FUNCTION_BLOCK Module_call
VAR_INPUT
END_VAR
VAR_OUTPUT
END_VAR
VAR
	CC1_UNIT1_3_Cyl: FB_CylinderModule;	
	CC2_UNIT2_3_Cyl: FB_CylinderModule;
	CC3_UNIT3_3_Cyl: FB_CylinderModule;
	CC4_UNIT4_3_Cyl: FB_CylinderModule;
	CC5_UNIT5_1_Cyl: FB_CylinderModule;
	CC6_UNIT6_1_Cyl: FB_CylinderModule;
	CC1_Feedback_FB: Feedback_FB;
	CC2_Feedback_FB: Feedback_FB;
	CC3_Feedback_FB: Feedback_FB;
	CC4_Feedback_FB: Feedback_FB;
	CC5_Feedback_FB: Feedback_FB;
	CC6_Feedback_FB: Feedback_FB;
	CC1_Feedback_1: BOOL;
	CC1_Feedback_2: BOOL;
	CC2_Feedback_1: BOOL;
	CC2_Feedback_2: BOOL;
	CC3_Feedback_1: BOOL;
	CC3_Feedback_2: BOOL;
	CC4_Feedback_1: BOOL;
	CC4_Feedback_2: BOOL;
	PowerOn: PowerOn;
	TurnTable_0: TurnTable;
	TT_Feedback_FB: Feedback_FB;
	Trunion_0: Trunion;
	Tr_Feedback_FB: Feedback_FB;
	RollerDoor_0: RollerDoor;
	Door_Feedback_FB: Feedback_FB;
	MH_Robot: Robot;
	Weld_Robot: Robot;
	Auto_Sequence_0: Auto_Sequence;
	TR_Feedback_FB1: Feedback_FB;
	HomeSequence_0: HomeSequence;
	Alarms_0: Alarms;
END_VAR
VAR // added by the converter: edge detectors and wires of the graphical bodies
    _w1, _w2, _w3, _w4, _w5, _w6, _w7, _w8 : BOOL;
END_VAR

// note: this text did not pass the execution check against the stored diagram
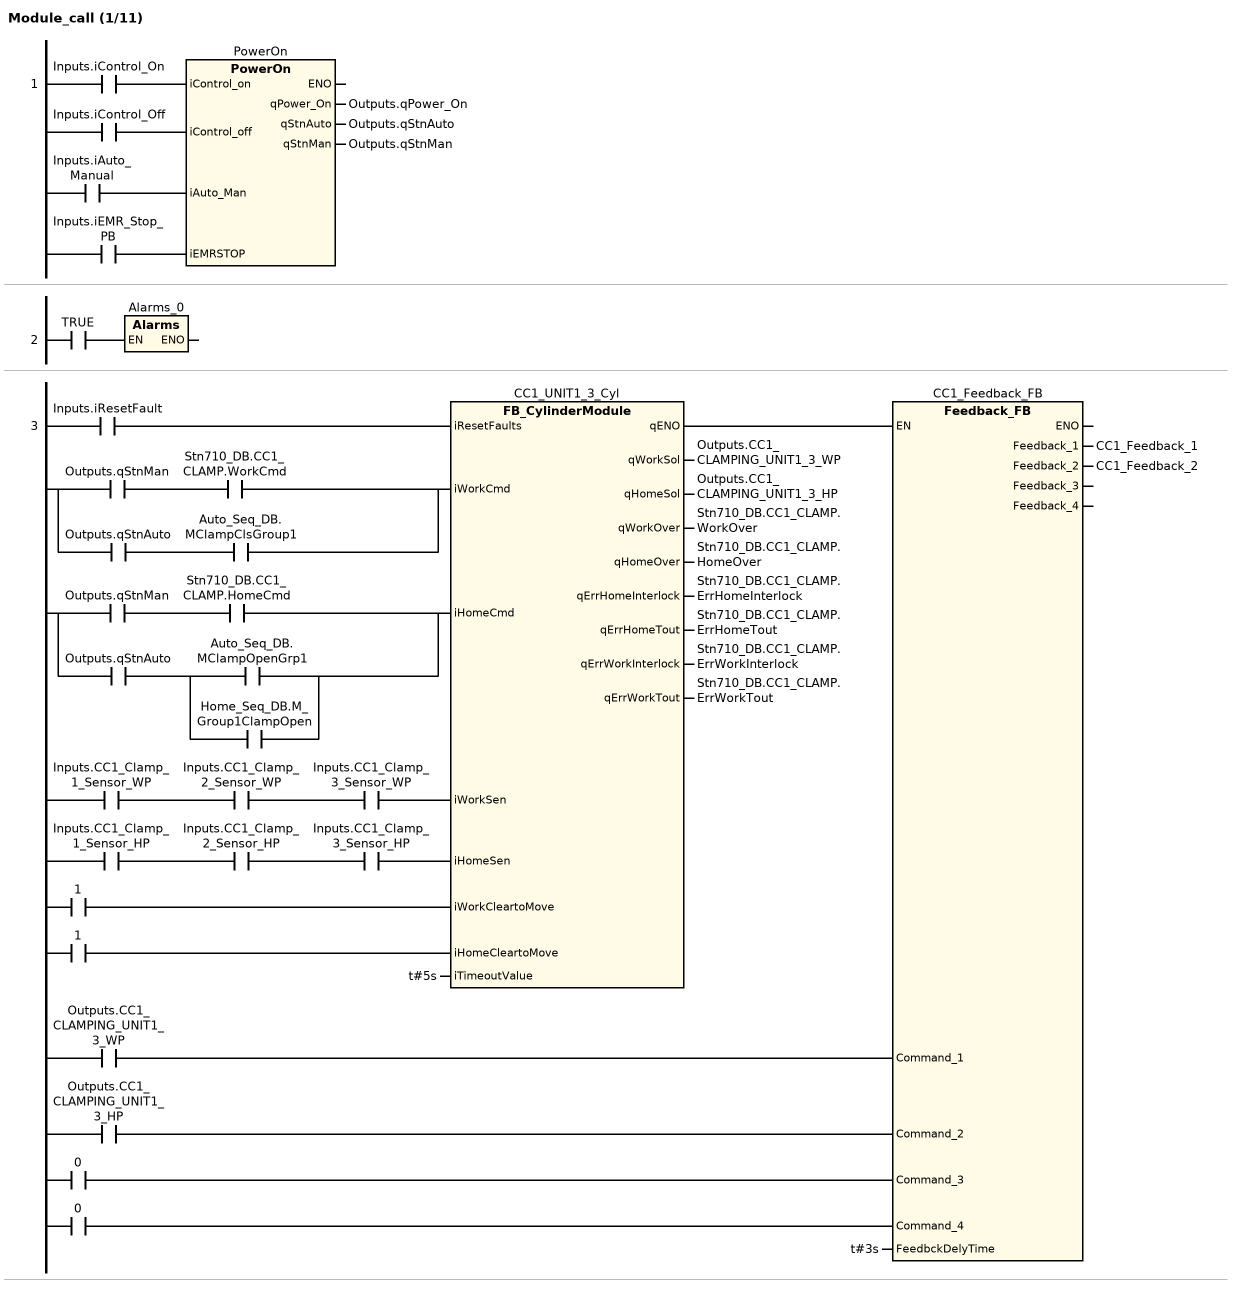
// NETWORK 1
PowerOn(
    iControl_on := Inputs.iControl_On,
    iControl_off := Inputs.iControl_Off,
    iAuto_Man := Inputs.iAuto_Manual,
    iEMRSTOP := Inputs.iEMR_Stop_PB,
    qPower_On => Outputs.qPower_On,
    qStnAuto => Outputs.qStnAuto,
    qStnMan => Outputs.qStnMan);

// NETWORK 2
Alarms_0(EN := TRUE); // Alarms

// NETWORK 3
CC1_UNIT1_3_Cyl(
    iResetFaults := Inputs.iResetFault,
    iWorkCmd := Outputs.qStnMan AND Stn710_DB.CC1_CLAMP.WorkCmd OR Outputs.qStnAuto AND Auto_Seq_DB.MClampClsGroup1,
    iHomeCmd := Outputs.qStnMan AND Stn710_DB.CC1_CLAMP.HomeCmd OR Outputs.qStnAuto AND (Auto_Seq_DB.MClampOpenGrp1 OR Home_Seq_DB.M_Group1ClampOpen),
    iWorkSen := Inputs.CC1_Clamp_1_Sensor_WP AND Inputs.CC1_Clamp_2_Sensor_WP AND Inputs.CC1_Clamp_3_Sensor_WP,
    iHomeSen := Inputs.CC1_Clamp_1_Sensor_HP AND Inputs.CC1_Clamp_2_Sensor_HP AND Inputs.CC1_Clamp_3_Sensor_HP,
    iWorkCleartoMove := 1,
    iHomeCleartoMove := 1,
    iTimeoutValue := t#5s,
    qWorkSol => Outputs.CC1_CLAMPING_UNIT1_3_WP,
    qHomeSol => Outputs.CC1_CLAMPING_UNIT1_3_HP,
    qWorkOver => Stn710_DB.CC1_CLAMP.WorkOver,
    qHomeOver => Stn710_DB.CC1_CLAMP.HomeOver,
    qErrHomeInterlock => Stn710_DB.CC1_CLAMP.ErrHomeInterlock,
    qErrHomeTout => Stn710_DB.CC1_CLAMP.ErrHomeTout,
    qErrWorkInterlock => Stn710_DB.CC1_CLAMP.ErrWorkInterlock,
    qErrWorkTout => Stn710_DB.CC1_CLAMP.ErrWorkTout); // FB_CylinderModule
CC1_Feedback_FB(
    EN := CC1_UNIT1_3_Cyl.qENO,
    Command_1 := Outputs.CC1_CLAMPING_UNIT1_3_WP,
    Command_2 := Outputs.CC1_CLAMPING_UNIT1_3_HP,
    Command_3 := 0,
    Command_4 := 0,
    FeedbckDelyTime := t#3s,
    Feedback_1 => CC1_Feedback_1,
    Feedback_2 => CC1_Feedback_2); // Feedback_FB

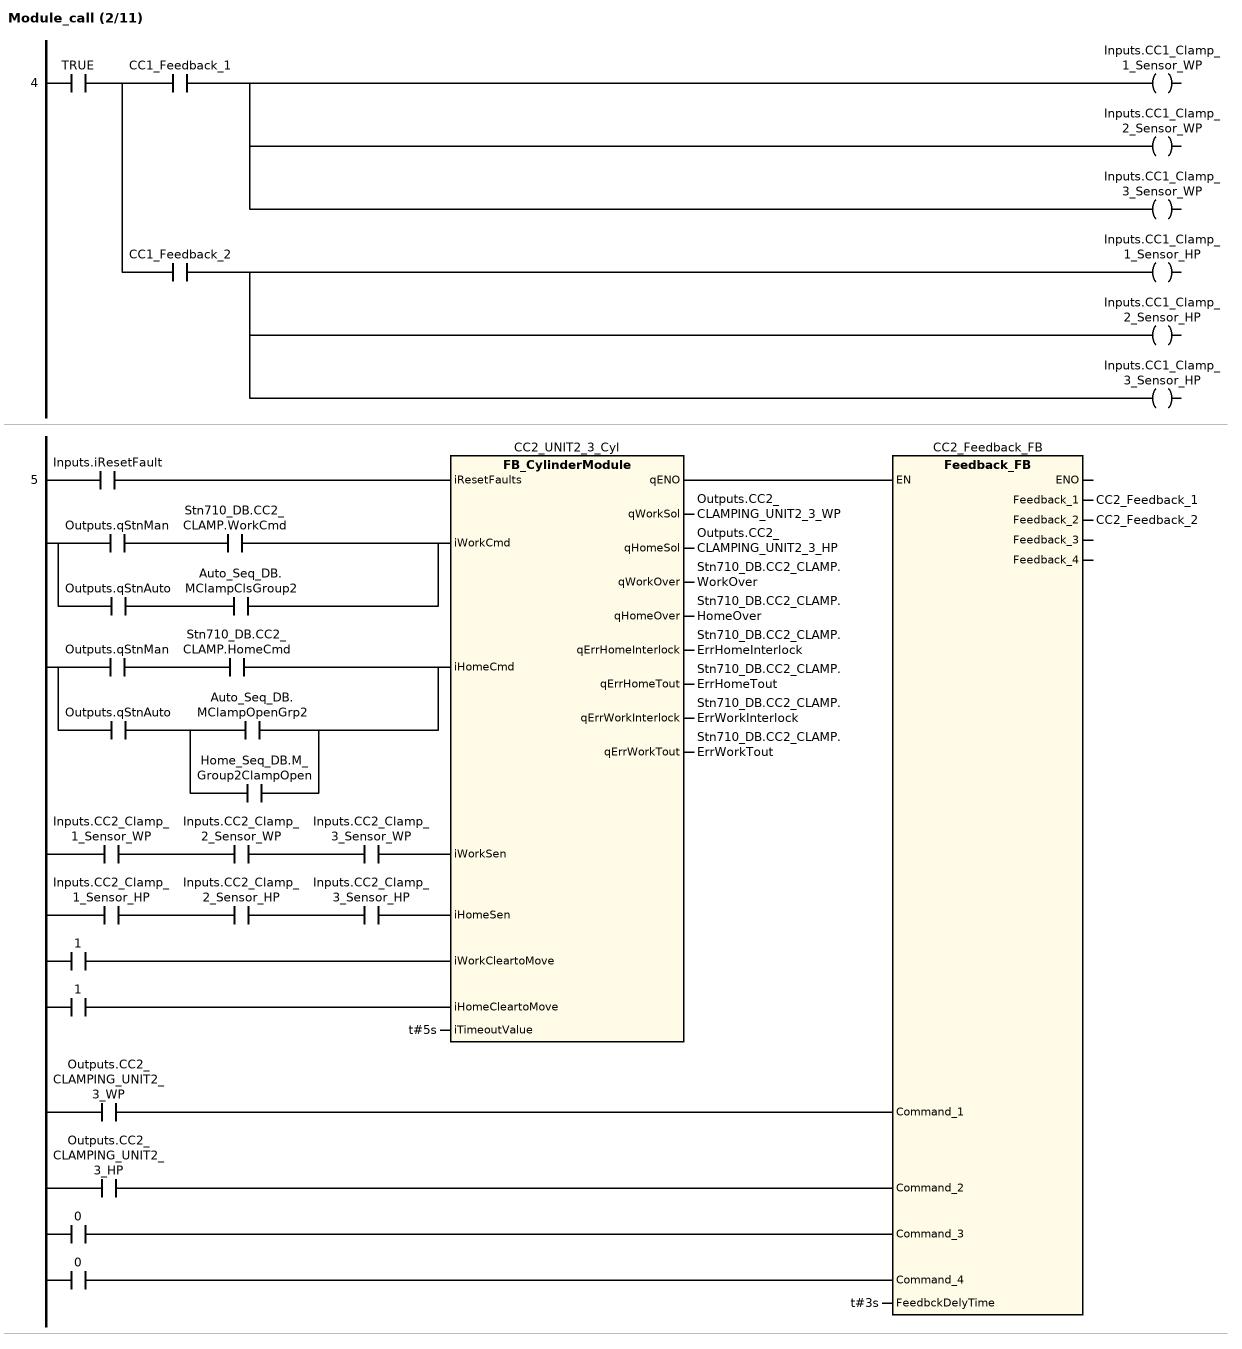
// NETWORK 4
_w1 := TRUE AND CC1_Feedback_1;
Inputs.CC1_Clamp_1_Sensor_WP := _w1;
Inputs.CC1_Clamp_2_Sensor_WP := _w1;
Inputs.CC1_Clamp_3_Sensor_WP := _w1;
_w2 := TRUE AND CC1_Feedback_2;
Inputs.CC1_Clamp_1_Sensor_HP := _w2;
Inputs.CC1_Clamp_2_Sensor_HP := _w2;
Inputs.CC1_Clamp_3_Sensor_HP := _w2;

// NETWORK 5
CC2_UNIT2_3_Cyl(
    iResetFaults := Inputs.iResetFault,
    iWorkCmd := Outputs.qStnMan AND Stn710_DB.CC2_CLAMP.WorkCmd OR Outputs.qStnAuto AND Auto_Seq_DB.MClampClsGroup2,
    iHomeCmd := Outputs.qStnMan AND Stn710_DB.CC2_CLAMP.HomeCmd OR Outputs.qStnAuto AND (Auto_Seq_DB.MClampOpenGrp2 OR Home_Seq_DB.M_Group2ClampOpen),
    iWorkSen := Inputs.CC2_Clamp_1_Sensor_WP AND Inputs.CC2_Clamp_2_Sensor_WP AND Inputs.CC2_Clamp_3_Sensor_WP,
    iHomeSen := Inputs.CC2_Clamp_1_Sensor_HP AND Inputs.CC2_Clamp_2_Sensor_HP AND Inputs.CC2_Clamp_3_Sensor_HP,
    iWorkCleartoMove := 1,
    iHomeCleartoMove := 1,
    iTimeoutValue := t#5s,
    qWorkSol => Outputs.CC2_CLAMPING_UNIT2_3_WP,
    qHomeSol => Outputs.CC2_CLAMPING_UNIT2_3_HP,
    qWorkOver => Stn710_DB.CC2_CLAMP.WorkOver,
    qHomeOver => Stn710_DB.CC2_CLAMP.HomeOver,
    qErrHomeInterlock => Stn710_DB.CC2_CLAMP.ErrHomeInterlock,
    qErrHomeTout => Stn710_DB.CC2_CLAMP.ErrHomeTout,
    qErrWorkInterlock => Stn710_DB.CC2_CLAMP.ErrWorkInterlock,
    qErrWorkTout => Stn710_DB.CC2_CLAMP.ErrWorkTout); // FB_CylinderModule
CC2_Feedback_FB(
    EN := CC2_UNIT2_3_Cyl.qENO,
    Command_1 := Outputs.CC2_CLAMPING_UNIT2_3_WP,
    Command_2 := Outputs.CC2_CLAMPING_UNIT2_3_HP,
    Command_3 := 0,
    Command_4 := 0,
    FeedbckDelyTime := t#3s,
    Feedback_1 => CC2_Feedback_1,
    Feedback_2 => CC2_Feedback_2); // Feedback_FB

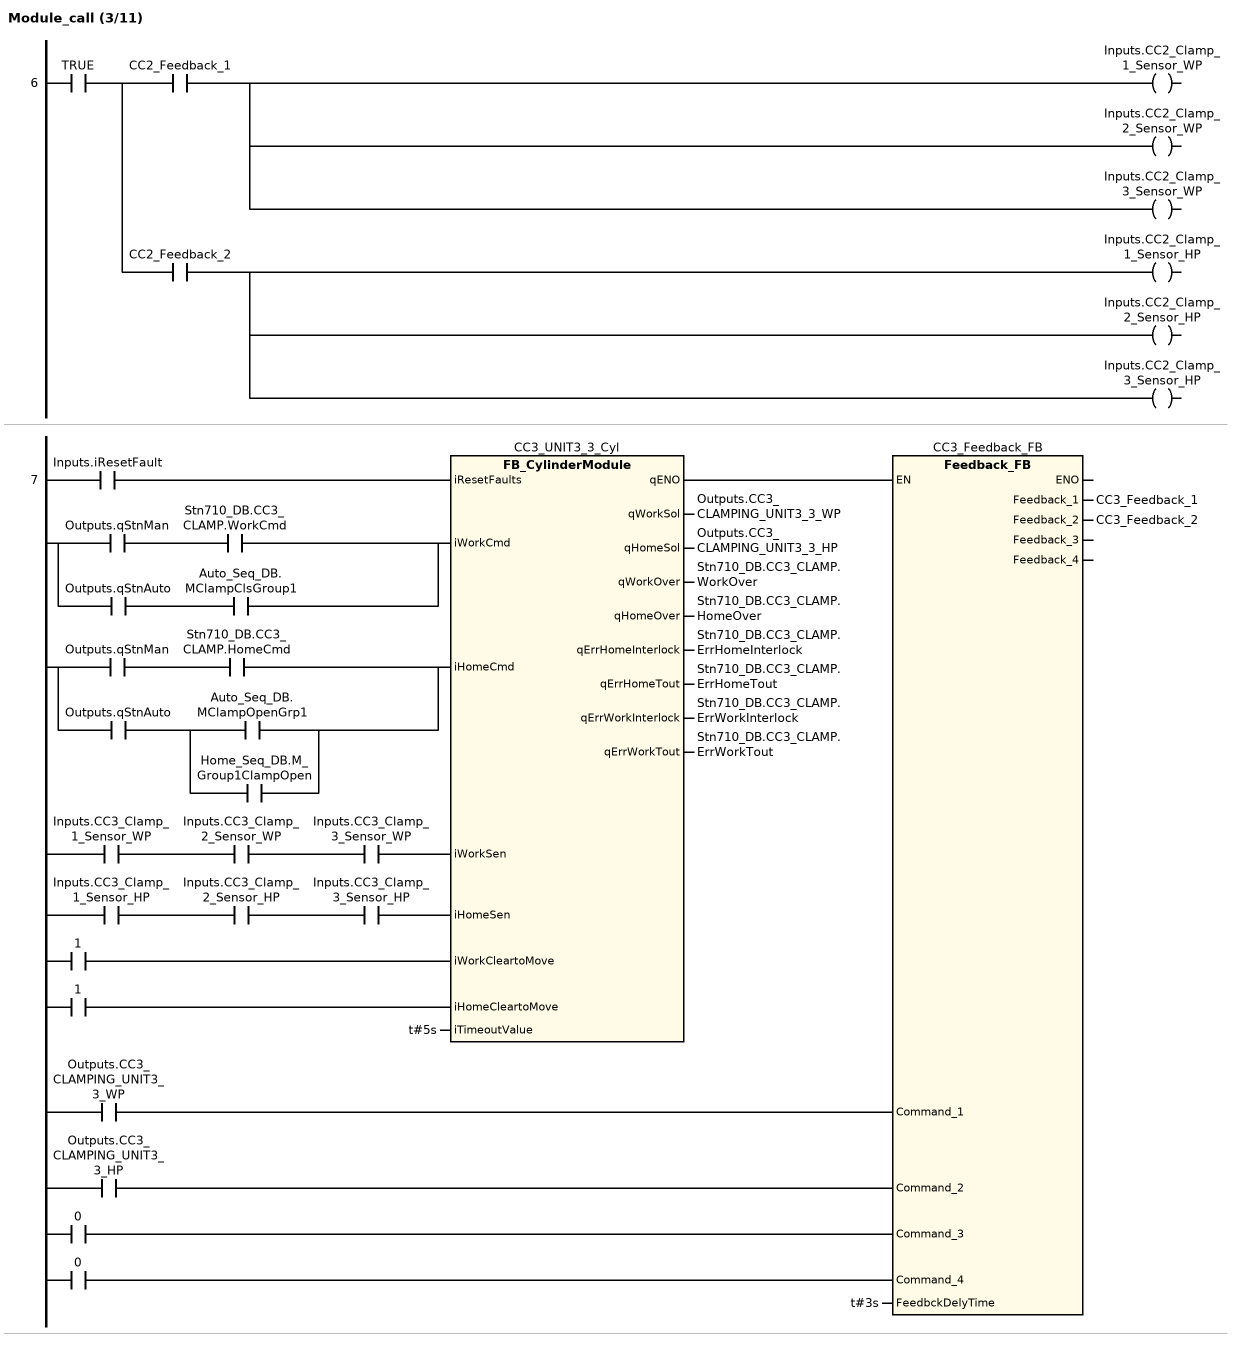
// NETWORK 6
_w3 := TRUE AND CC2_Feedback_1;
Inputs.CC2_Clamp_1_Sensor_WP := _w3;
Inputs.CC2_Clamp_2_Sensor_WP := _w3;
Inputs.CC2_Clamp_3_Sensor_WP := _w3;
_w4 := TRUE AND CC2_Feedback_2;
Inputs.CC2_Clamp_1_Sensor_HP := _w4;
Inputs.CC2_Clamp_2_Sensor_HP := _w4;
Inputs.CC2_Clamp_3_Sensor_HP := _w4;

// NETWORK 7
CC3_UNIT3_3_Cyl(
    iResetFaults := Inputs.iResetFault,
    iWorkCmd := Outputs.qStnMan AND Stn710_DB.CC3_CLAMP.WorkCmd OR Outputs.qStnAuto AND Auto_Seq_DB.MClampClsGroup1,
    iHomeCmd := Outputs.qStnMan AND Stn710_DB.CC3_CLAMP.HomeCmd OR Outputs.qStnAuto AND (Auto_Seq_DB.MClampOpenGrp1 OR Home_Seq_DB.M_Group1ClampOpen),
    iWorkSen := Inputs.CC3_Clamp_1_Sensor_WP AND Inputs.CC3_Clamp_2_Sensor_WP AND Inputs.CC3_Clamp_3_Sensor_WP,
    iHomeSen := Inputs.CC3_Clamp_1_Sensor_HP AND Inputs.CC3_Clamp_2_Sensor_HP AND Inputs.CC3_Clamp_3_Sensor_HP,
    iWorkCleartoMove := 1,
    iHomeCleartoMove := 1,
    iTimeoutValue := t#5s,
    qWorkSol => Outputs.CC3_CLAMPING_UNIT3_3_WP,
    qHomeSol => Outputs.CC3_CLAMPING_UNIT3_3_HP,
    qWorkOver => Stn710_DB.CC3_CLAMP.WorkOver,
    qHomeOver => Stn710_DB.CC3_CLAMP.HomeOver,
    qErrHomeInterlock => Stn710_DB.CC3_CLAMP.ErrHomeInterlock,
    qErrHomeTout => Stn710_DB.CC3_CLAMP.ErrHomeTout,
    qErrWorkInterlock => Stn710_DB.CC3_CLAMP.ErrWorkInterlock,
    qErrWorkTout => Stn710_DB.CC3_CLAMP.ErrWorkTout); // FB_CylinderModule
CC3_Feedback_FB(
    EN := CC3_UNIT3_3_Cyl.qENO,
    Command_1 := Outputs.CC3_CLAMPING_UNIT3_3_WP,
    Command_2 := Outputs.CC3_CLAMPING_UNIT3_3_HP,
    Command_3 := 0,
    Command_4 := 0,
    FeedbckDelyTime := t#3s,
    Feedback_1 => CC3_Feedback_1,
    Feedback_2 => CC3_Feedback_2); // Feedback_FB

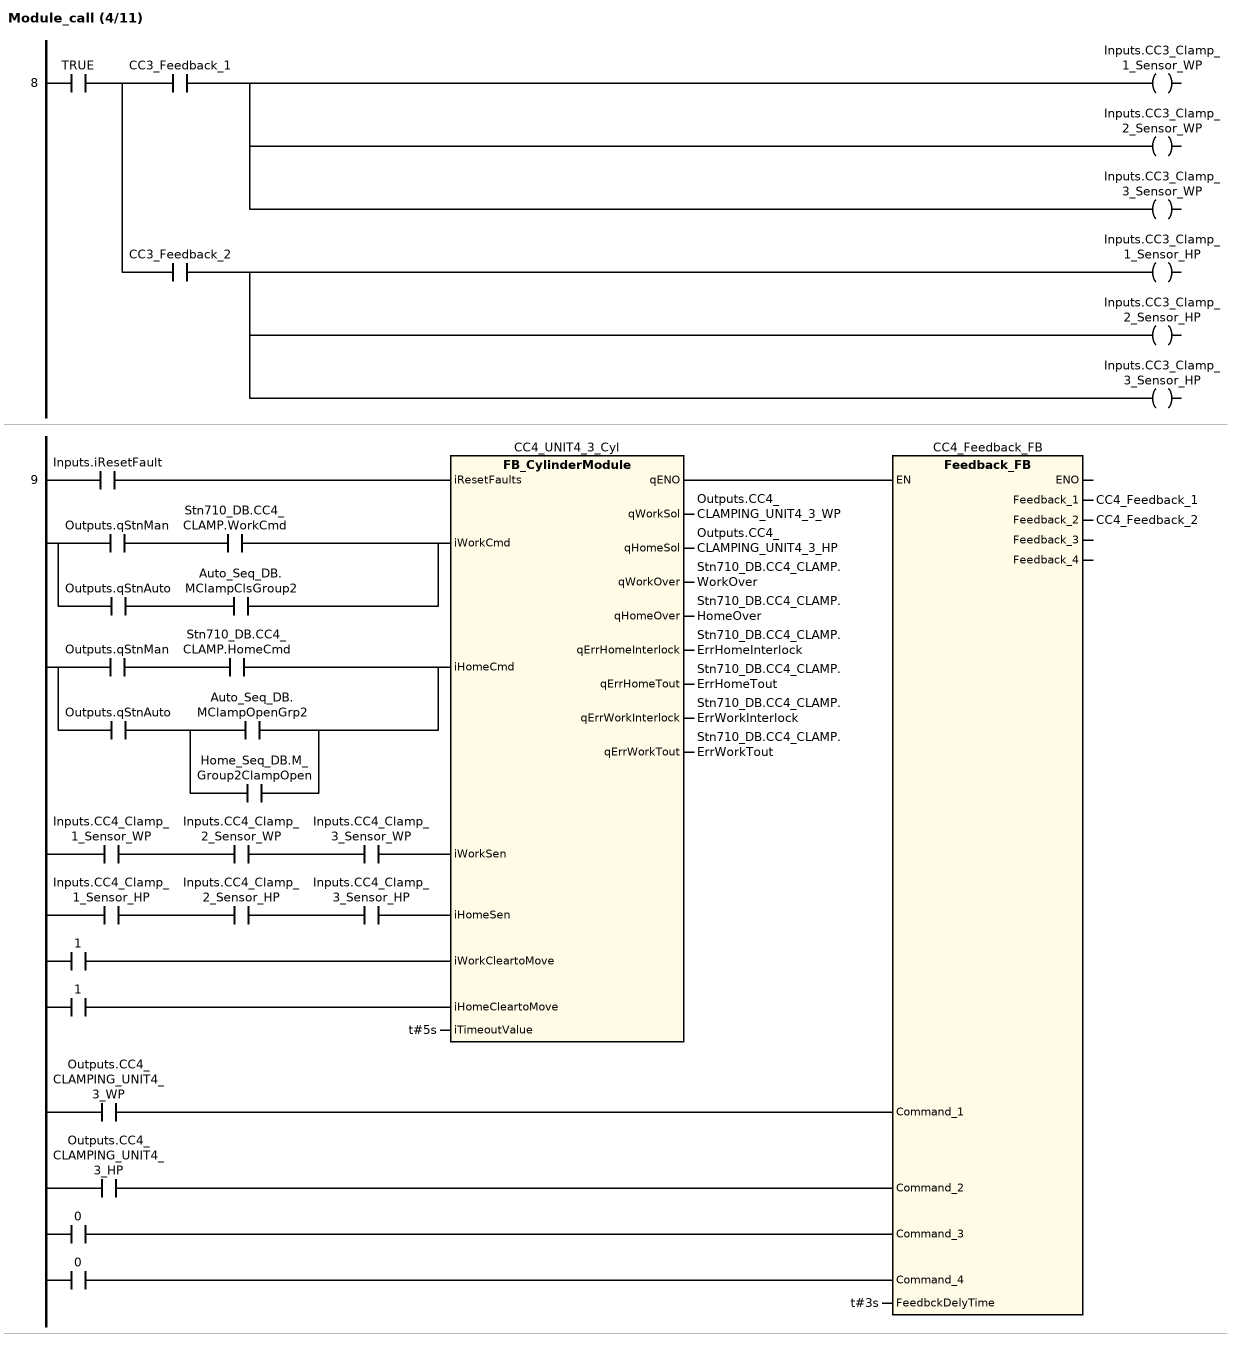
// NETWORK 8
_w5 := TRUE AND CC3_Feedback_1;
Inputs.CC3_Clamp_1_Sensor_WP := _w5;
Inputs.CC3_Clamp_2_Sensor_WP := _w5;
Inputs.CC3_Clamp_3_Sensor_WP := _w5;
_w6 := TRUE AND CC3_Feedback_2;
Inputs.CC3_Clamp_1_Sensor_HP := _w6;
Inputs.CC3_Clamp_2_Sensor_HP := _w6;
Inputs.CC3_Clamp_3_Sensor_HP := _w6;

// NETWORK 9
CC4_UNIT4_3_Cyl(
    iResetFaults := Inputs.iResetFault,
    iWorkCmd := Outputs.qStnMan AND Stn710_DB.CC4_CLAMP.WorkCmd OR Outputs.qStnAuto AND Auto_Seq_DB.MClampClsGroup2,
    iHomeCmd := Outputs.qStnMan AND Stn710_DB.CC4_CLAMP.HomeCmd OR Outputs.qStnAuto AND (Auto_Seq_DB.MClampOpenGrp2 OR Home_Seq_DB.M_Group2ClampOpen),
    iWorkSen := Inputs.CC4_Clamp_1_Sensor_WP AND Inputs.CC4_Clamp_2_Sensor_WP AND Inputs.CC4_Clamp_3_Sensor_WP,
    iHomeSen := Inputs.CC4_Clamp_1_Sensor_HP AND Inputs.CC4_Clamp_2_Sensor_HP AND Inputs.CC4_Clamp_3_Sensor_HP,
    iWorkCleartoMove := 1,
    iHomeCleartoMove := 1,
    iTimeoutValue := t#5s,
    qWorkSol => Outputs.CC4_CLAMPING_UNIT4_3_WP,
    qHomeSol => Outputs.CC4_CLAMPING_UNIT4_3_HP,
    qWorkOver => Stn710_DB.CC4_CLAMP.WorkOver,
    qHomeOver => Stn710_DB.CC4_CLAMP.HomeOver,
    qErrHomeInterlock => Stn710_DB.CC4_CLAMP.ErrHomeInterlock,
    qErrHomeTout => Stn710_DB.CC4_CLAMP.ErrHomeTout,
    qErrWorkInterlock => Stn710_DB.CC4_CLAMP.ErrWorkInterlock,
    qErrWorkTout => Stn710_DB.CC4_CLAMP.ErrWorkTout); // FB_CylinderModule
CC4_Feedback_FB(
    EN := CC4_UNIT4_3_Cyl.qENO,
    Command_1 := Outputs.CC4_CLAMPING_UNIT4_3_WP,
    Command_2 := Outputs.CC4_CLAMPING_UNIT4_3_HP,
    Command_3 := 0,
    Command_4 := 0,
    FeedbckDelyTime := t#3s,
    Feedback_1 => CC4_Feedback_1,
    Feedback_2 => CC4_Feedback_2); // Feedback_FB

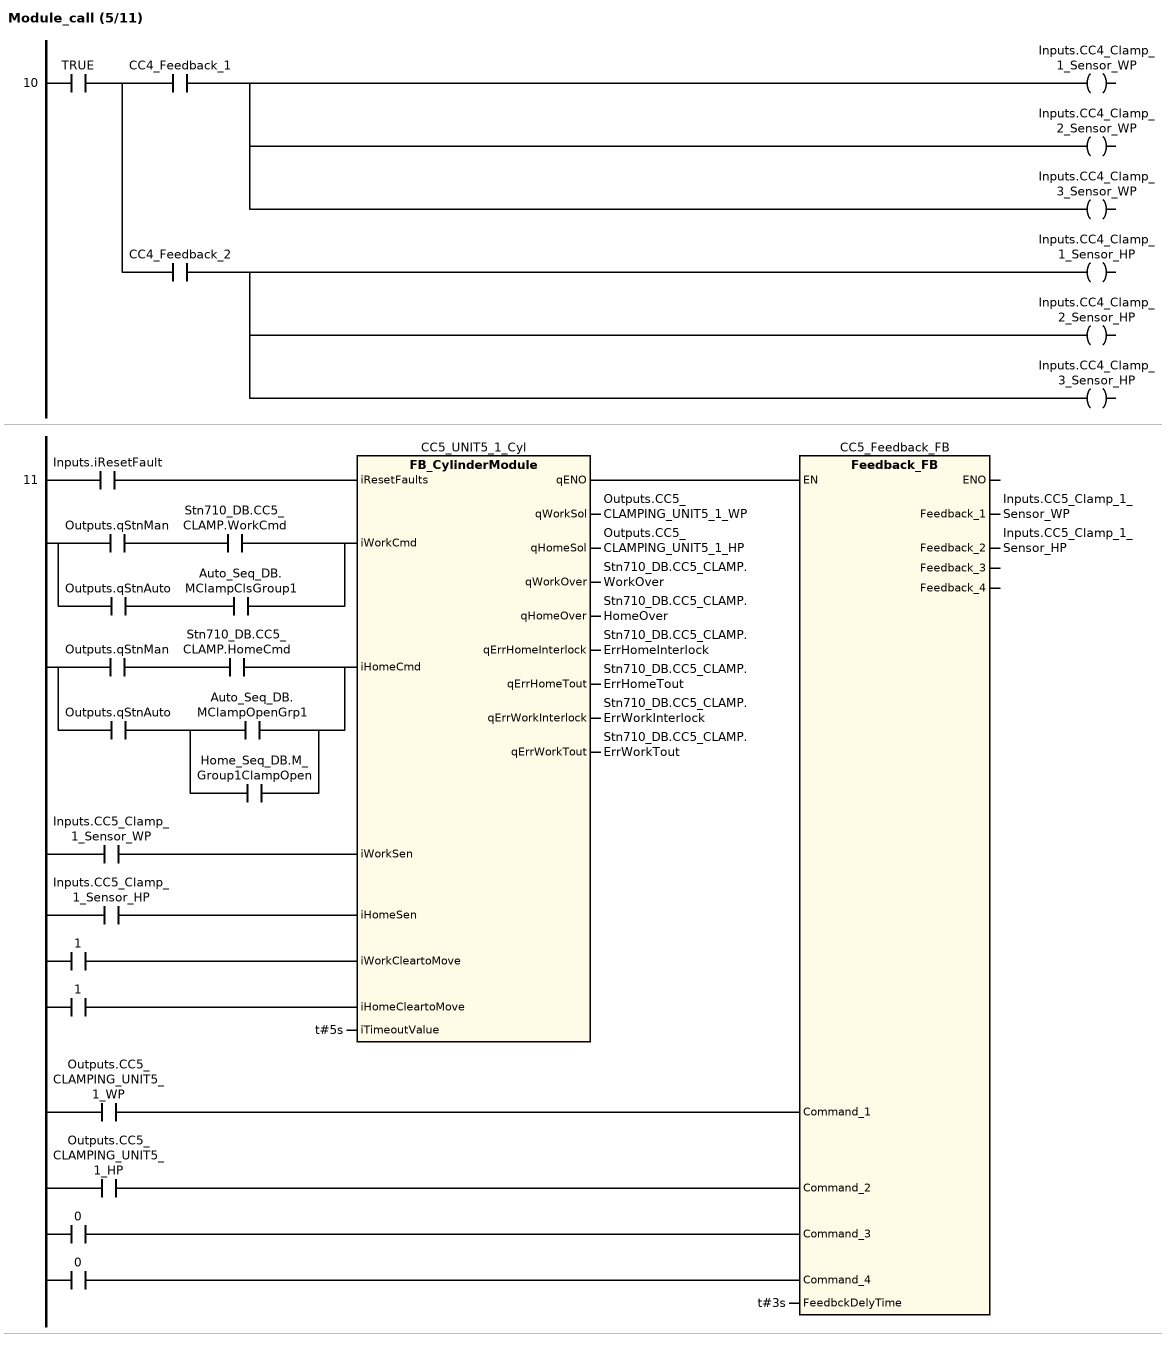
// NETWORK 10
_w7 := TRUE AND CC4_Feedback_1;
Inputs.CC4_Clamp_1_Sensor_WP := _w7;
Inputs.CC4_Clamp_2_Sensor_WP := _w7;
Inputs.CC4_Clamp_3_Sensor_WP := _w7;
_w8 := TRUE AND CC4_Feedback_2;
Inputs.CC4_Clamp_1_Sensor_HP := _w8;
Inputs.CC4_Clamp_2_Sensor_HP := _w8;
Inputs.CC4_Clamp_3_Sensor_HP := _w8;

// NETWORK 11
CC5_UNIT5_1_Cyl(
    iResetFaults := Inputs.iResetFault,
    iWorkCmd := Outputs.qStnMan AND Stn710_DB.CC5_CLAMP.WorkCmd OR Outputs.qStnAuto AND Auto_Seq_DB.MClampClsGroup1,
    iHomeCmd := Outputs.qStnMan AND Stn710_DB.CC5_CLAMP.HomeCmd OR Outputs.qStnAuto AND (Auto_Seq_DB.MClampOpenGrp1 OR Home_Seq_DB.M_Group1ClampOpen),
    iWorkSen := Inputs.CC5_Clamp_1_Sensor_WP,
    iHomeSen := Inputs.CC5_Clamp_1_Sensor_HP,
    iWorkCleartoMove := 1,
    iHomeCleartoMove := 1,
    iTimeoutValue := t#5s,
    qWorkSol => Outputs.CC5_CLAMPING_UNIT5_1_WP,
    qHomeSol => Outputs.CC5_CLAMPING_UNIT5_1_HP,
    qWorkOver => Stn710_DB.CC5_CLAMP.WorkOver,
    qHomeOver => Stn710_DB.CC5_CLAMP.HomeOver,
    qErrHomeInterlock => Stn710_DB.CC5_CLAMP.ErrHomeInterlock,
    qErrHomeTout => Stn710_DB.CC5_CLAMP.ErrHomeTout,
    qErrWorkInterlock => Stn710_DB.CC5_CLAMP.ErrWorkInterlock,
    qErrWorkTout => Stn710_DB.CC5_CLAMP.ErrWorkTout); // FB_CylinderModule
CC5_Feedback_FB(
    EN := CC5_UNIT5_1_Cyl.qENO,
    Command_1 := Outputs.CC5_CLAMPING_UNIT5_1_WP,
    Command_2 := Outputs.CC5_CLAMPING_UNIT5_1_HP,
    Command_3 := 0,
    Command_4 := 0,
    FeedbckDelyTime := t#3s,
    Feedback_1 => Inputs.CC5_Clamp_1_Sensor_WP,
    Feedback_2 => Inputs.CC5_Clamp_1_Sensor_HP); // Feedback_FB

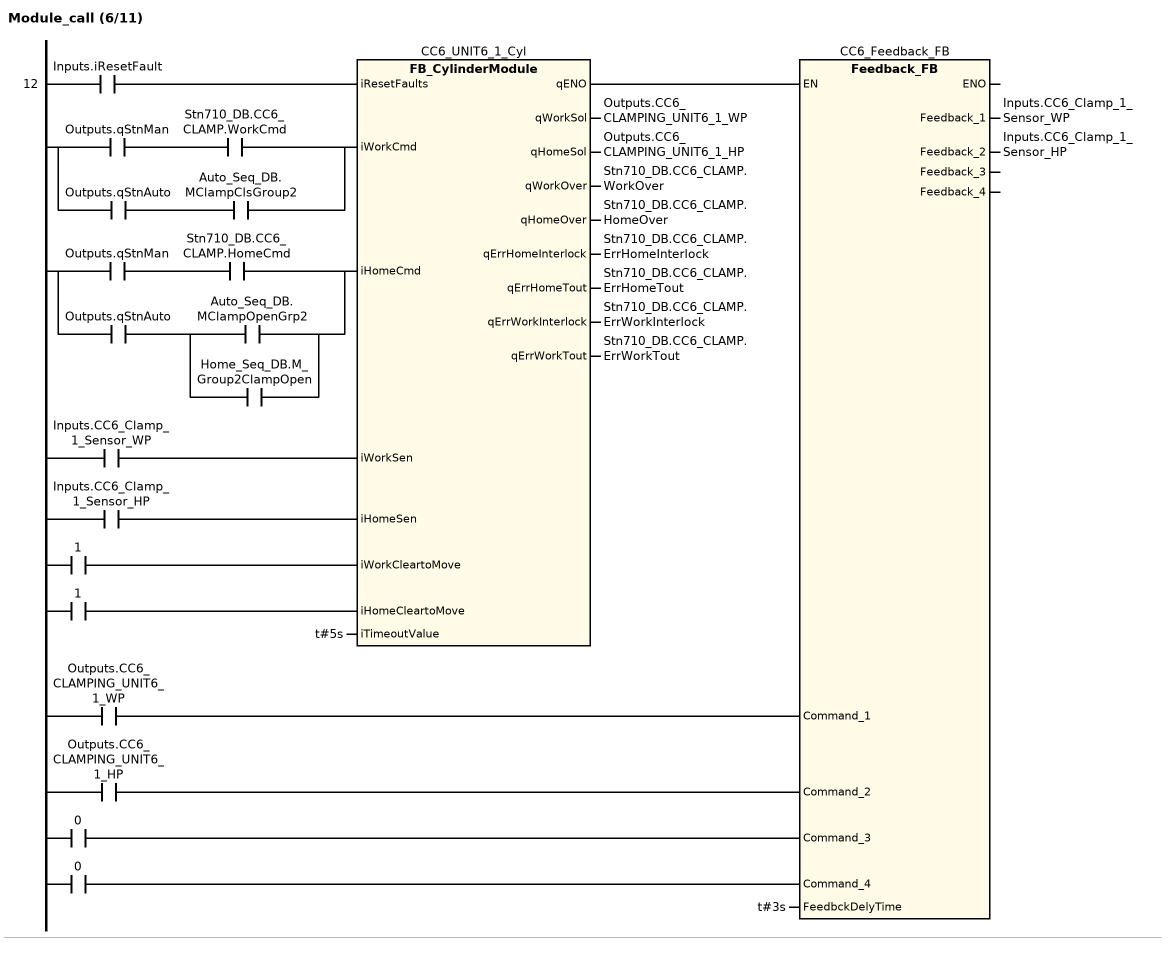
// NETWORK 12
CC6_UNIT6_1_Cyl(
    iResetFaults := Inputs.iResetFault,
    iWorkCmd := Outputs.qStnMan AND Stn710_DB.CC6_CLAMP.WorkCmd OR Outputs.qStnAuto AND Auto_Seq_DB.MClampClsGroup2,
    iHomeCmd := Outputs.qStnMan AND Stn710_DB.CC6_CLAMP.HomeCmd OR Outputs.qStnAuto AND (Auto_Seq_DB.MClampOpenGrp2 OR Home_Seq_DB.M_Group2ClampOpen),
    iWorkSen := Inputs.CC6_Clamp_1_Sensor_WP,
    iHomeSen := Inputs.CC6_Clamp_1_Sensor_HP,
    iWorkCleartoMove := 1,
    iHomeCleartoMove := 1,
    iTimeoutValue := t#5s,
    qWorkSol => Outputs.CC6_CLAMPING_UNIT6_1_WP,
    qHomeSol => Outputs.CC6_CLAMPING_UNIT6_1_HP,
    qWorkOver => Stn710_DB.CC6_CLAMP.WorkOver,
    qHomeOver => Stn710_DB.CC6_CLAMP.HomeOver,
    qErrHomeInterlock => Stn710_DB.CC6_CLAMP.ErrHomeInterlock,
    qErrHomeTout => Stn710_DB.CC6_CLAMP.ErrHomeTout,
    qErrWorkInterlock => Stn710_DB.CC6_CLAMP.ErrWorkInterlock,
    qErrWorkTout => Stn710_DB.CC6_CLAMP.ErrWorkTout); // FB_CylinderModule
CC6_Feedback_FB(
    EN := CC6_UNIT6_1_Cyl.qENO,
    Command_1 := Outputs.CC6_CLAMPING_UNIT6_1_WP,
    Command_2 := Outputs.CC6_CLAMPING_UNIT6_1_HP,
    Command_3 := 0,
    Command_4 := 0,
    FeedbckDelyTime := t#3s,
    Feedback_1 => Inputs.CC6_Clamp_1_Sensor_WP,
    Feedback_2 => Inputs.CC6_Clamp_1_Sensor_HP); // Feedback_FB

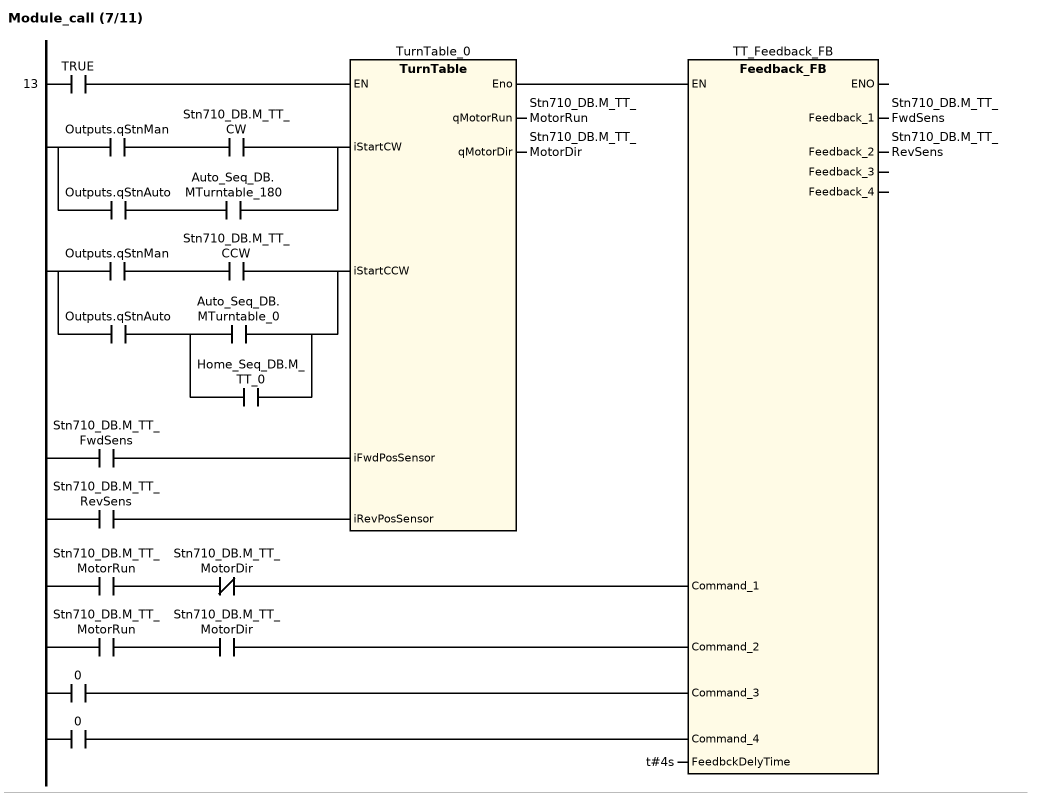
// NETWORK 13
TurnTable_0(
    EN := TRUE,
    iStartCW := Outputs.qStnMan AND Stn710_DB.M_TT_CW OR Outputs.qStnAuto AND Auto_Seq_DB.MTurntable_180,
    iStartCCW := Outputs.qStnMan AND Stn710_DB.M_TT_CCW OR Outputs.qStnAuto AND (Auto_Seq_DB.MTurntable_0 OR Home_Seq_DB.M_TT_0),
    iFwdPosSensor := Stn710_DB.M_TT_FwdSens,
    iRevPosSensor := Stn710_DB.M_TT_RevSens,
    qMotorRun => Stn710_DB.M_TT_MotorRun,
    qMotorDir => Stn710_DB.M_TT_MotorDir); // TurnTable
TT_Feedback_FB(
    EN := TRUE,
    Command_1 := Stn710_DB.M_TT_MotorRun AND NOT Stn710_DB.M_TT_MotorDir,
    Command_2 := Stn710_DB.M_TT_MotorRun AND Stn710_DB.M_TT_MotorDir,
    Command_3 := 0,
    Command_4 := 0,
    FeedbckDelyTime := t#4s,
    Feedback_1 => Stn710_DB.M_TT_FwdSens,
    Feedback_2 => Stn710_DB.M_TT_RevSens); // Feedback_FB

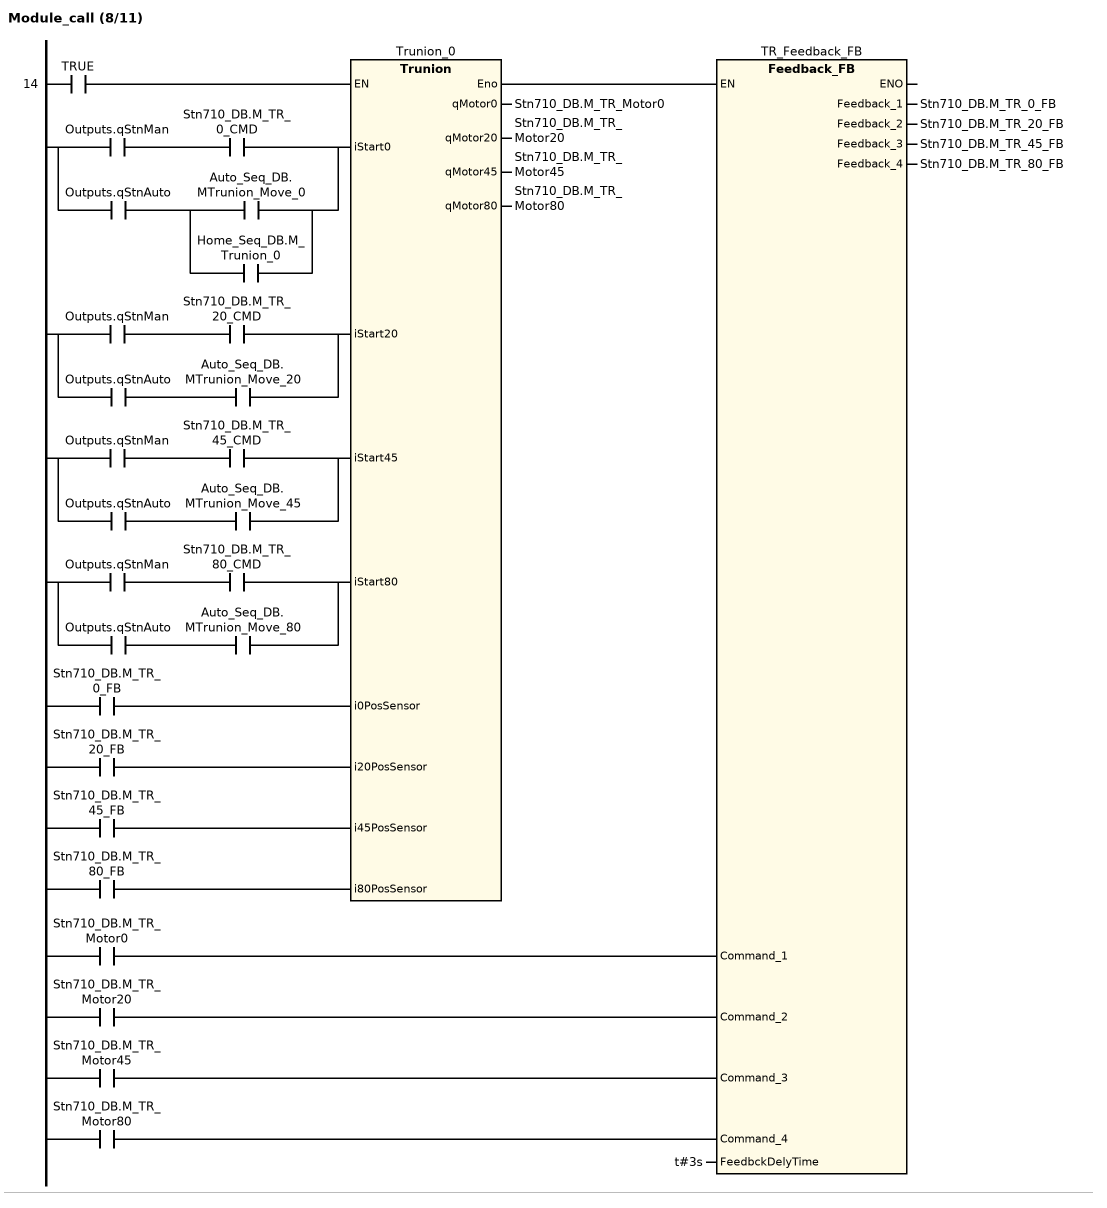
// NETWORK 14
Trunion_0(
    EN := TRUE,
    iStart0 := Outputs.qStnMan AND Stn710_DB.M_TR_0_CMD OR Outputs.qStnAuto AND (Auto_Seq_DB.MTrunion_Move_0 OR Home_Seq_DB.M_Trunion_0),
    iStart20 := Outputs.qStnMan AND Stn710_DB.M_TR_20_CMD OR Outputs.qStnAuto AND Auto_Seq_DB.MTrunion_Move_20,
    iStart45 := Outputs.qStnMan AND Stn710_DB.M_TR_45_CMD OR Outputs.qStnAuto AND Auto_Seq_DB.MTrunion_Move_45,
    iStart80 := Outputs.qStnMan AND Stn710_DB.M_TR_80_CMD OR Outputs.qStnAuto AND Auto_Seq_DB.MTrunion_Move_80,
    i0PosSensor := Stn710_DB.M_TR_0_FB,
    i20PosSensor := Stn710_DB.M_TR_20_FB,
    i45PosSensor := Stn710_DB.M_TR_45_FB,
    i80PosSensor := Stn710_DB.M_TR_80_FB,
    qMotor0 => Stn710_DB.M_TR_Motor0,
    qMotor20 => Stn710_DB.M_TR_Motor20,
    qMotor45 => Stn710_DB.M_TR_Motor45,
    qMotor80 => Stn710_DB.M_TR_Motor80); // Trunion
TR_Feedback_FB(
    EN := TRUE,
    Command_1 := Stn710_DB.M_TR_Motor0,
    Command_2 := Stn710_DB.M_TR_Motor20,
    Command_3 := Stn710_DB.M_TR_Motor45,
    Command_4 := Stn710_DB.M_TR_Motor80,
    FeedbckDelyTime := t#3s,
    Feedback_1 => Stn710_DB.M_TR_0_FB,
    Feedback_2 => Stn710_DB.M_TR_20_FB,
    Feedback_3 => Stn710_DB.M_TR_45_FB,
    Feedback_4 => Stn710_DB.M_TR_80_FB); // Feedback_FB

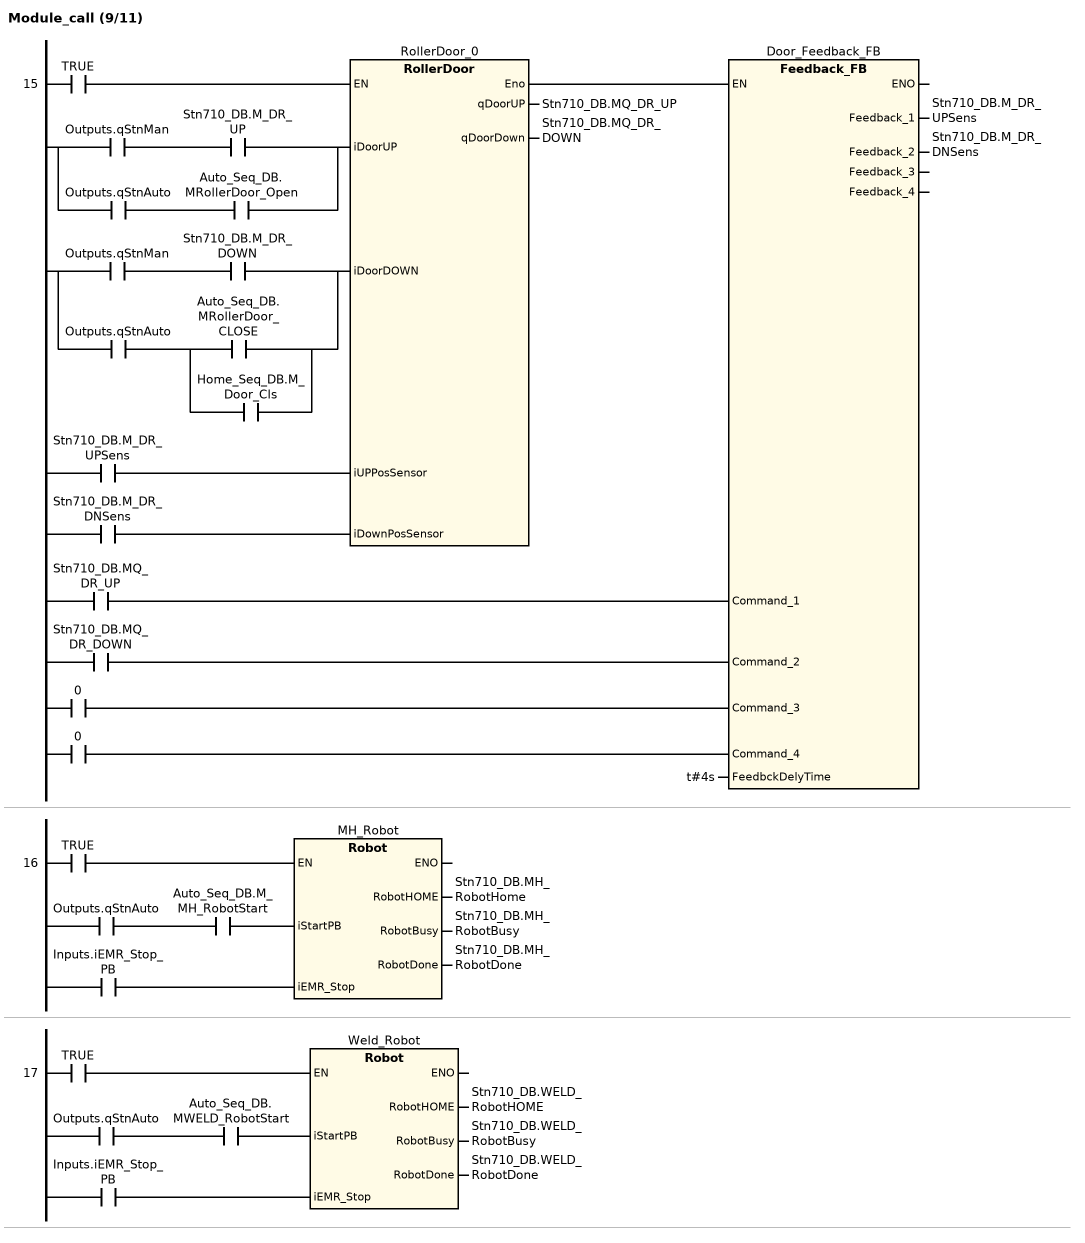
// NETWORK 15
RollerDoor_0(
    EN := TRUE,
    iDoorUP := Outputs.qStnMan AND Stn710_DB.M_DR_UP OR Outputs.qStnAuto AND Auto_Seq_DB.MRollerDoor_Open,
    iDoorDOWN := Outputs.qStnMan AND Stn710_DB.M_DR_DOWN OR Outputs.qStnAuto AND (Auto_Seq_DB.MRollerDoor_CLOSE OR Home_Seq_DB.M_Door_Cls),
    iUPPosSensor := Stn710_DB.M_DR_UPSens,
    iDownPosSensor := Stn710_DB.M_DR_DNSens,
    qDoorUP => Stn710_DB.MQ_DR_UP,
    qDoorDown => Stn710_DB.MQ_DR_DOWN); // RollerDoor
Door_Feedback_FB(
    EN := TRUE,
    Command_1 := Stn710_DB.MQ_DR_UP,
    Command_2 := Stn710_DB.MQ_DR_DOWN,
    Command_3 := 0,
    Command_4 := 0,
    FeedbckDelyTime := t#4s,
    Feedback_1 => Stn710_DB.M_DR_UPSens,
    Feedback_2 => Stn710_DB.M_DR_DNSens); // Feedback_FB

// NETWORK 16
MH_Robot(
    EN := TRUE,
    iStartPB := Outputs.qStnAuto AND Auto_Seq_DB.M_MH_RobotStart,
    iEMR_Stop := Inputs.iEMR_Stop_PB,
    RobotHOME => Stn710_DB.MH_RobotHome,
    RobotBusy => Stn710_DB.MH_RobotBusy,
    RobotDone => Stn710_DB.MH_RobotDone); // Robot

// NETWORK 17
Weld_Robot(
    EN := TRUE,
    iStartPB := Outputs.qStnAuto AND Auto_Seq_DB.MWELD_RobotStart,
    iEMR_Stop := Inputs.iEMR_Stop_PB,
    RobotHOME => Stn710_DB.WELD_RobotHOME,
    RobotBusy => Stn710_DB.WELD_RobotBusy,
    RobotDone => Stn710_DB.WELD_RobotDone); // Robot

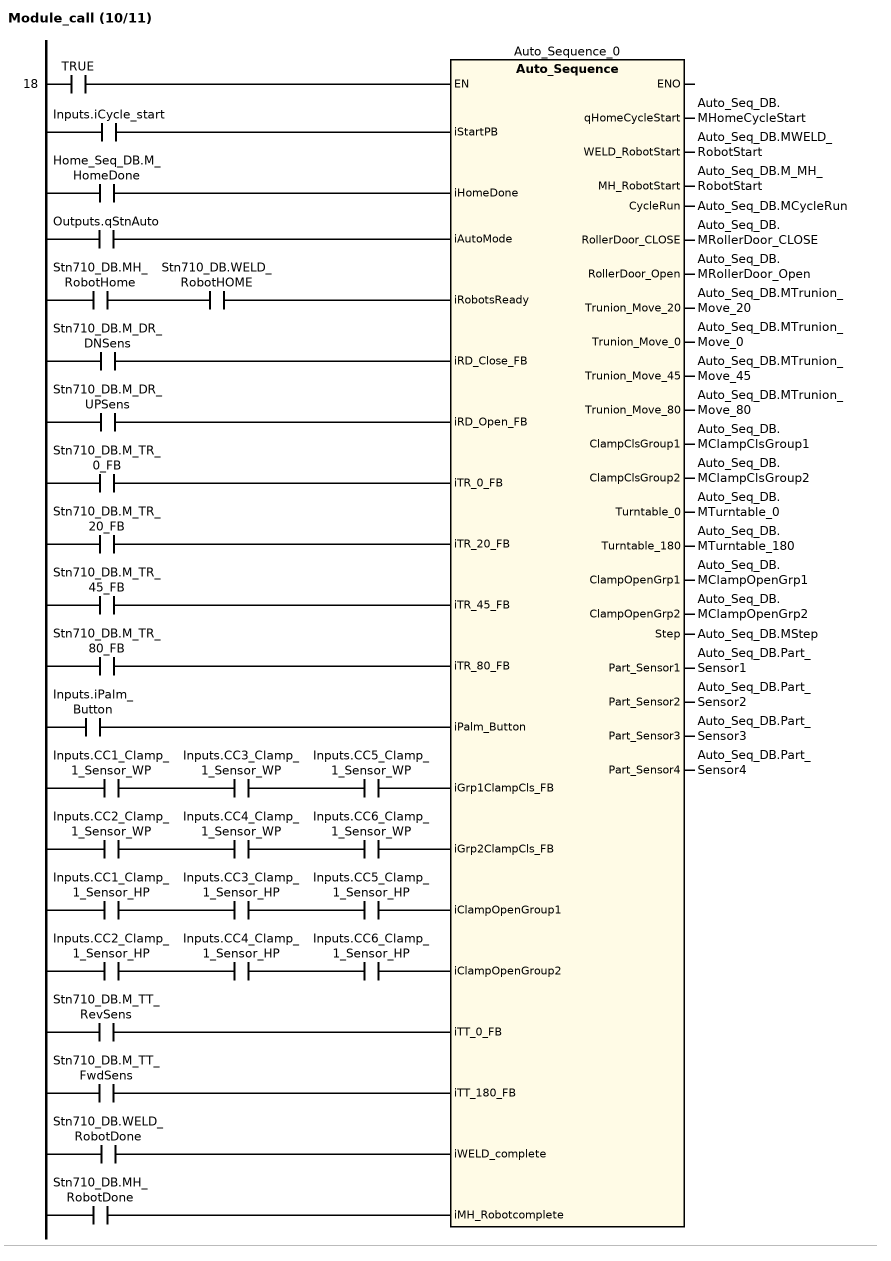
// NETWORK 18
Auto_Sequence_0(
    EN := TRUE,
    iStartPB := Inputs.iCycle_start,
    iHomeDone := Home_Seq_DB.M_HomeDone,
    iAutoMode := Outputs.qStnAuto,
    iRobotsReady := Stn710_DB.MH_RobotHome AND Stn710_DB.WELD_RobotHOME,
    iRD_Close_FB := Stn710_DB.M_DR_DNSens,
    iRD_Open_FB := Stn710_DB.M_DR_UPSens,
    iTR_0_FB := Stn710_DB.M_TR_0_FB,
    iTR_20_FB := Stn710_DB.M_TR_20_FB,
    iTR_45_FB := Stn710_DB.M_TR_45_FB,
    iTR_80_FB := Stn710_DB.M_TR_80_FB,
    iPalm_Button := Inputs.iPalm_Button,
    iGrp1ClampCls_FB := Inputs.CC1_Clamp_1_Sensor_WP AND Inputs.CC3_Clamp_1_Sensor_WP AND Inputs.CC5_Clamp_1_Sensor_WP,
    iGrp2ClampCls_FB := Inputs.CC2_Clamp_1_Sensor_WP AND Inputs.CC4_Clamp_1_Sensor_WP AND Inputs.CC6_Clamp_1_Sensor_WP,
    iClampOpenGroup1 := Inputs.CC1_Clamp_1_Sensor_HP AND Inputs.CC3_Clamp_1_Sensor_HP AND Inputs.CC5_Clamp_1_Sensor_HP,
    iClampOpenGroup2 := Inputs.CC2_Clamp_1_Sensor_HP AND Inputs.CC4_Clamp_1_Sensor_HP AND Inputs.CC6_Clamp_1_Sensor_HP,
    iTT_0_FB := Stn710_DB.M_TT_RevSens,
    iTT_180_FB := Stn710_DB.M_TT_FwdSens,
    iWELD_complete := Stn710_DB.WELD_RobotDone,
    iMH_Robotcomplete := Stn710_DB.MH_RobotDone,
    qHomeCycleStart => Auto_Seq_DB.MHomeCycleStart,
    WELD_RobotStart => Auto_Seq_DB.MWELD_RobotStart,
    MH_RobotStart => Auto_Seq_DB.M_MH_RobotStart,
    CycleRun => Auto_Seq_DB.MCycleRun,
    RollerDoor_CLOSE => Auto_Seq_DB.MRollerDoor_CLOSE,
    RollerDoor_Open => Auto_Seq_DB.MRollerDoor_Open,
    Trunion_Move_20 => Auto_Seq_DB.MTrunion_Move_20,
    Trunion_Move_0 => Auto_Seq_DB.MTrunion_Move_0,
    Trunion_Move_45 => Auto_Seq_DB.MTrunion_Move_45,
    Trunion_Move_80 => Auto_Seq_DB.MTrunion_Move_80,
    ClampClsGroup1 => Auto_Seq_DB.MClampClsGroup1,
    ClampClsGroup2 => Auto_Seq_DB.MClampClsGroup2,
    Turntable_0 => Auto_Seq_DB.MTurntable_0,
    Turntable_180 => Auto_Seq_DB.MTurntable_180,
    ClampOpenGrp1 => Auto_Seq_DB.MClampOpenGrp1,
    ClampOpenGrp2 => Auto_Seq_DB.MClampOpenGrp2,
    Step => Auto_Seq_DB.MStep,
    Part_Sensor1 => Auto_Seq_DB.Part_Sensor1,
    Part_Sensor2 => Auto_Seq_DB.Part_Sensor2,
    Part_Sensor3 => Auto_Seq_DB.Part_Sensor3,
    Part_Sensor4 => Auto_Seq_DB.Part_Sensor4); // Auto_Sequence

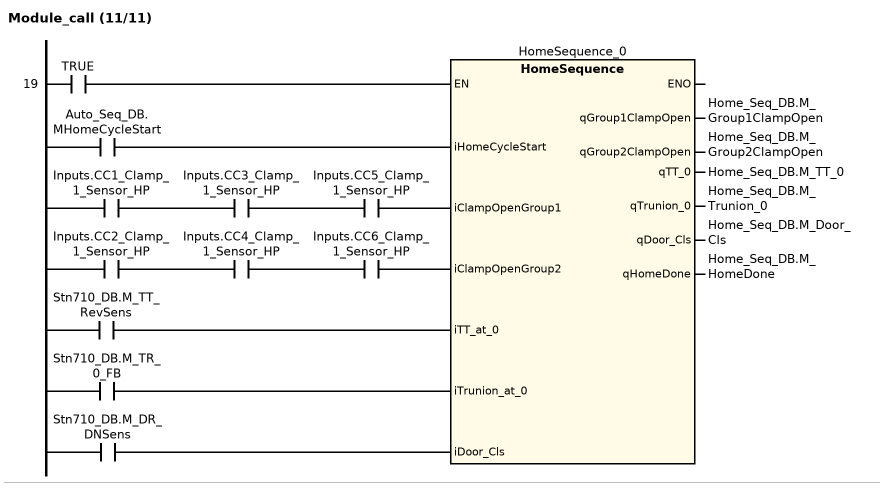
// NETWORK 19
HomeSequence_0(
    EN := TRUE,
    iHomeCycleStart := Auto_Seq_DB.MHomeCycleStart,
    iClampOpenGroup1 := Inputs.CC1_Clamp_1_Sensor_HP AND Inputs.CC3_Clamp_1_Sensor_HP AND Inputs.CC5_Clamp_1_Sensor_HP,
    iClampOpenGroup2 := Inputs.CC2_Clamp_1_Sensor_HP AND Inputs.CC4_Clamp_1_Sensor_HP AND Inputs.CC6_Clamp_1_Sensor_HP,
    iTT_at_0 := Stn710_DB.M_TT_RevSens,
    iTrunion_at_0 := Stn710_DB.M_TR_0_FB,
    iDoor_Cls := Stn710_DB.M_DR_DNSens,
    qGroup1ClampOpen => Home_Seq_DB.M_Group1ClampOpen,
    qGroup2ClampOpen => Home_Seq_DB.M_Group2ClampOpen,
    qTT_0 => Home_Seq_DB.M_TT_0,
    qTrunion_0 => Home_Seq_DB.M_Trunion_0,
    qDoor_Cls => Home_Seq_DB.M_Door_Cls,
    qHomeDone => Home_Seq_DB.M_HomeDone); // HomeSequence

END_FUNCTION_BLOCK

(* stored: Version 1.1.0.1, ProductVersion 3.1.4024.16
   POU Module_call: Id {0fabfa72-1626-4a34-917e-e1c074627036}, SpecialFunc None *)
